(* IEC 61131-3 sources: plc_on_fpga_riscv_hybrid/RV_FPGA_PLC_IDE_Projects/Timer_Test_2, 1 file *)

(* ---- Timer_Test_2.il ---- *)
VAR
    Elapsed_Time   : TIME
    Preset_Time   : TIME
    TON_0   : TON
END_VAR

PROGRAM Timer_Test_2
    R1 :
        LD     T#1500ms
        ST     Preset_Time
        CAL TON_0(
            IN := %SW.0,
            PT := Preset_Time,
            ET => Elapsed_Time,
            Q  => %LEDR.0)
END_PROGRAM
